FUNCTION_BLOCK WStrMem
VAR_INPUT
END_VAR
VAR_OUTPUT
END_VAR
VAR
	mem : WSTRING;
END_VAR

METHOD APPEND : BOOL
VAR_INPUT
	STR : WSTRING;
END_VAR
mem := WCONCAT(mem , STR);
END_METHOD

METHOD INSERT : BOOL
VAR_INPUT
	STR : WSTRING;
END_VAR
mem := WCONCAT(STR, mem);
END_METHOD

PROPERTY READ : WSTRING
GET
READ := mem;
END_GET
END_PROPERTY

METHOD WRITE : BOOL
VAR_INPUT
	STR :WSTRING;
END_VAR
mem := STR;
END_METHOD

END_FUNCTION_BLOCK

(* stored: Version 1.1.0.1, ProductVersion 3.1.4026.13
   POU WStrMem: Id {57b8977a-b7cb-4c5e-afc6-7fec4c45060c}, SpecialFunc None
   Method APPEND: Id {495be183-616f-46de-8cad-3f3417a8abe3}
   Method INSERT: Id {3c051e22-732d-4f3a-b6c6-1d4276a7bb12}
   Property READ: Id {34841f93-1a9a-4d7a-badc-56f58fbe476e}
   Get Get: Id {12555e73-c774-4905-b09e-f475937de223}
   Method WRITE: Id {ad5ff546-3031-4f6b-89b5-e2c5a16fb975} *)
